Yaskawa INFORM job: R1_W23(-90,90)(KAMERA)KM-OK.JBI

/JOB
//NAME R1_W23(-90,90)(KAMERA)KM-OK
///FOLDERNAME KRIS-SCIANA
//POS
///NPOS 55,55,0,5,0,0
///TOOL 0
///POSTYPE PULSE
///PULSE
C00000=-89180,31382,-23952,-16361,97536,59278
C00001=-17295,-105465,-106227,-19833,67209,69782
C00002=-8987,30952,-6160,-16006,80817,78065
C00003=-6788,-10602,-33117,-24212,62605,65754
C00004=-163140,-11215,-34889,-20382,57885,63547
C00005=-203904,-58095,-46309,10621,38304,46048
C00006=-203487,-40393,-28240,10719,36271,46001
C00007=-203487,-40393,-28240,10719,36271,46001
C00008=-203959,-38853,-27279,11114,36529,45767
C00009=-203487,-40393,-28240,10719,36271,46001
C00010=-203487,-40209,-27675,10783,36024,45965
C00011=-203487,-40393,-28240,10719,36271,46001
C00012=-192128,-45410,-37586,851,40249,51912
C00013=-140490,-42544,-36309,-37655,52482,75470
C00014=-143651,-39413,-29798,-37339,49183,75221
C00015=-145177,-37980,-27379,-36985,47916,74946
C00016=-145177,-37586,-26135,-37291,47462,75153
C00017=-145177,-37980,-27379,-36985,47916,74946
C00018=-146306,-37306,-26950,-36367,47499,74504
C00019=-145177,-37980,-27379,-36985,47916,74946
C00020=-138763,-52848,-44323,-38599,52956,76175
C00021=-154433,-43630,-61410,25728,86407,75332
C00022=-157641,-41809,-45369,39510,82356,72747
C00023=-148492,-37514,-30679,46567,75096,74143
C00024=-147977,-37344,-29960,46625,75219,74031
C00025=-147977,-36975,-28647,46735,74787,73821
C00026=-147977,-37344,-29960,46625,75219,74031
C00027=-146918,-38035,-30399,46516,74609,74261
C00028=-147977,-37344,-29960,46625,75219,74031
C00029=-153021,-35361,-33920,46660,79630,74096
C00030=-152320,-32341,-31934,46536,79496,74375
C00031=-146989,-36196,-28492,46503,73846,74285
C00032=-146989,-36196,-28492,46503,73846,74285
C00033=-146368,-36591,-28746,46432,73491,74420
C00034=-146989,-36196,-28492,46503,73846,74285
C00035=-146989,-36005,-27823,46564,73626,74177
C00036=-146989,-36196,-28492,46503,73846,74285
C00037=-156146,-31178,-34336,46806,82942,74156
C00038=-173128,-58148,-60869,24512,63483,63733
C00039=-203904,-58095,-46309,10621,38304,46048
C00040=-226839,-42186,-16856,66354,38232,28633
C00041=-226839,-42186,-16856,66354,38232,28633
C00042=-206322,-31295,-10155,54911,26194,36153
C00043=-187832,-8667,6108,29122,18400,49604
C00044=-173150,-5234,-8709,-16783,43253,61887
C00045=-219674,-82383,-78158,21046,47819,39959
C00046=-139475,-34778,-60414,43000,96089,79010
C00047=-142954,-57885,-47199,43086,82851,71938
C00048=-129499,-44465,-33619,42620,63719,77920
C00049=-132687,-61427,-28566,69264,45165,61174
C00050=-129900,-31757,-11692,64398,45403,64574
C00051=-127366,15735,25677,62559,44442,65932
C00052=-128866,12122,12330,57798,48673,68999
C00053=-129695,34239,15315,39996,71522,81230
C00054=-131597,15649,-11680,39434,77876,82839
BC00000=287918,15031,1075171
BC00001=6401,8474,1075170
BC00002=22330,1815,1075164
BC00003=16324,8003,1075175
BC00004=398174,7783,1075175
BC00005=398174,134143,1075175
BC00006=398174,134144,1075172
BC00007=398174,134144,1075172
BC00008=398174,134144,1075172
BC00009=398174,134144,1075172
BC00010=398174,134144,1075172
BC00011=398174,134144,1075172
BC00012=390479,134144,1075172
BC00013=314704,134144,1075172
BC00014=314704,134144,1075172
BC00015=314704,134144,1075172
BC00016=314704,134144,1075172
BC00017=314704,134144,1075172
BC00018=314704,134144,1075172
BC00019=314704,134144,1075172
BC00020=314704,134144,1075172
BC00021=241815,134144,1075232
BC00022=226895,134144,1075172
BC00023=226895,134144,1075172
BC00024=226895,134144,1075172
BC00025=226895,134144,1075172
BC00026=226895,134144,1075172
BC00027=226895,134144,1075172
BC00028=226895,134144,1075172
BC00029=226895,134144,1075172
BC00030=226895,59489,1075172
BC00031=226895,59489,1075172
BC00032=226895,59489,1075172
BC00033=226895,59489,1075172
BC00034=226895,59489,1075172
BC00035=226895,59489,1075172
BC00036=226895,59489,1075172
BC00037=226895,59489,1075172
BC00038=312739,96905,1075174
BC00039=398174,134143,1075175
BC00040=398174,141900,1075175
BC00041=398174,141900,1075175
BC00042=398174,141900,1075175
BC00043=398174,141900,1075175
BC00044=398174,141900,1075175
BC00045=398174,141900,1075175
BC00046=194821,53250,1075175
BC00047=194821,53250,1075175
BC00048=194821,53250,1075175
BC00049=194821,53250,1075175
BC00050=194821,53250,1075175
BC00051=194821,53250,1075175
BC00052=194821,53250,1075175
BC00053=194821,53250,1075175
BC00054=194821,53250,1075175
///POSTYPE BASE
///RECTAN
///RCONF 0,0,0,0,1,0,0,0,0,0,0,0,0,0,0,0,0,0,0,0,0,0,0,0
P00006=2.006,1.622,-0.565,0.0000,0.0000,0.0000
P00021=0.073,2.058,-0.109,0.0000,0.0000,0.0000
P00022=2.006,1.622,-0.565,0.0000,0.0000,0.0000
///RCONF 0,0,0,0,0,0,0,0,0,0,0,0,0,0,0,0,0,0,0,0,0,0,0,0
P00023=-2.957,-4.083,2.762,0.0000,0.0000,0.0000
P00024=-1.466,-0.226,-0.419,0.0000,0.0000,0.0000
//INST
///DATE 2025/04/28 12:39
///ATTR SC,RW
///GROUP1 RB1,BS1
NOP
'r1_W23(-90,90)(kamera)
'Path W869
SFTOF
MOVJ C00000 BC00000 VJ=100.00
MOVJ C00001 BC00001 VJ=100.00
MOVJ C00002 BC00002 VJ=50.00
CALL JOB:CLEAN-R1_LONG
MOVJ C00003 BC00003 VJ=100.00
MOVJ C00004 BC00004 VJ=100.00
MOVJ C00005 BC00005 VJ=100.00
MOVJ C00006 BC00006 VJ=100.00
'POMIAR
MOVL C00007 BC00007 V=60.0
REFP 3 C00008 BC00008
CALL JOB:SEARCH-R1
SET P021 P006
SFTON P021
MOVL C00009 BC00009 V=60.0
REFP 3 C00010 BC00010
CALL JOB:SEARCH-R1
SET P021 P006
SFTON P021
MOVL C00011 BC00011 V=60.0
MOVJ C00012 BC00012 VJ=100.00
SFTOF
MOVJ C00013 BC00013 VJ=100.00
MOVJ C00014 BC00014 VJ=100.00
MOVL C00015 BC00015 V=60.0
REFP 3 C00016 BC00016
CALL JOB:SEARCH-R1
SET P022 P006
SFTON P022
MOVL C00017 BC00017 V=60.0
REFP 3 C00018 BC00018
CALL JOB:SEARCH-R1
SET P022 P006
SFTON P022
MOVL C00019 BC00019 V=60.0
MOVJ C00020 BC00020 VJ=100.00
SFTOF
MOVJ C00021 BC00021 VJ=100.00
MOVJ C00022 BC00022 VJ=100.00
MOVJ C00023 BC00023 VJ=100.00
MOVL C00024 BC00024 V=60.0
REFP 3 C00025 BC00025
CALL JOB:SEARCH-R1
SET P023 P006
SFTON P023
MOVL C00026 BC00026 V=60.0
REFP 3 C00027 BC00027
CALL JOB:SEARCH-R1
SET P023 P006
SFTON P023
MOVL C00028 BC00028 V=60.0
MOVJ C00029 BC00029 VJ=100.00
SFTOF
MOVJ C00030 BC00030 VJ=100.00
MOVJ C00031 BC00031 VJ=100.00
MOVL C00032 BC00032 V=60.0
REFP 3 C00033 BC00033
CALL JOB:SEARCH-R1
SET P024 P006
SFTON P024
MOVL C00034 BC00034 V=60.0
REFP 3 C00035 BC00035
CALL JOB:SEARCH-R1
SET P024 P006
SFTON P024
MOVL C00036 BC00036 V=60.0
MOVJ C00037 BC00037 VJ=100.00
MOVJ C00038 BC00038 VJ=100.00
SFTOF
CALL JOB:COFNIJ_DRUT
MOVJ C00039 BC00039 VJ=100.00
SFTON P021
COMM MOVJ C00040 BC00040 VJ=100.00
MOVL C00041 BC00041 V=666.7
MACRO1 MJ#(0) ARGF9
ARCON
SFTON P022
MOVL C00042 BC00042 V=9.2
MOVL C00043 BC00043 V=9.2
ARCOF
SFTOF
MOVL C00044 BC00044 V=166.7
MOVJ C00045 BC00045 VJ=100.00
MOVJ C00046 BC00046 VJ=100.00
'SPOINA2
MOVJ C00047 BC00047 VJ=100.00
SFTON P024
COMM MOVJ C00048 BC00048 VJ=15.00
MOVL C00049 BC00049 V=666.7 PL=0
MACRO1 MJ#(0) ARGF9
ARCON
SFTON P023
MOVL C00050 BC00050 V=9.2
MOVL C00051 BC00051 V=9.2
ARCOF
SFTOF
MOVL C00052 BC00052 V=666.7
MOVJ C00053 BC00053 VJ=100.00
MOVJ C00054 BC00054 VJ=100.00
END
